% RSLogix 500 project Sample1.RSS, saved by version 9.00.00.04 %
PROJECT "SAMPLE1"    % processor: Bul.1763 MicroLogix 1100 Series A %

PROGRAM FILES
  LAD 2 "MAIN"  21 rungs
  LAD 3 "D INPUT"  11 rungs
  LAD 4 "A INPUT"  66 rungs
  LAD 5 "D OUTPUT"  8 rungs
  LAD 6 "A OUTPUT"  21 rungs
  LAD 7 "ALARMS"  598 rungs
  LAD 8 "HMI IO"  323 rungs
  LAD 9 "LOOPS"  21 rungs
  LAD 10 "CONTROL"  80 rungs

DATA FILES
  O0 OUTPUT  4 elements
  I1 INPUT  6 elements
  S2 STATUS  66 elements
  B3 BINARY  100 elements
  T4 TIMER  256 elements
  C5 COUNTER  1 elements
  R6 CONTROL  1 elements
  N7 INTEGER  256 elements
  F8 FLOAT  249 elements
  B9 ALARMS  40 elements
  F10 F-SETPTS 1  256 elements
  N11 N-SETPTS 1  256 elements
  N12 PIDBLOCKS1  233 elements
  N13 DONOTTOUCH  128 elements
  N14 PIDBLOCKS2  233 elements
  N15 PIDBLOCKS3  143 elements
  B16 SYSCTRLS  10 elements
  T17 TIMERS 2  10 elements
  F18 F-SETPTS 2  93 elements
  N19 N-SETPTS 2  6 elements
  N20 MB_CFG  1 elements
  N21 MB_BIN  46 elements
  F22 MB_FLT1  256 elements
  F23 MB_FLT2  256 elements
  F24 MB_FLT3  256 elements
  F25 MB_FLT4  256 elements
  F26 MB_FLT5  256 elements
  F27 MB_FLT6  256 elements
  F28 MB_FLT7  256 elements
  F29 LAST_VAL1  256 elements
  F30 LAST_VAL2  256 elements
  F31 LAST_VAL3  256 elements
  N90 CH1 Diag  256 elements
  N91 CH0 Diag  32 elements

LADDER 2 "MAIN"
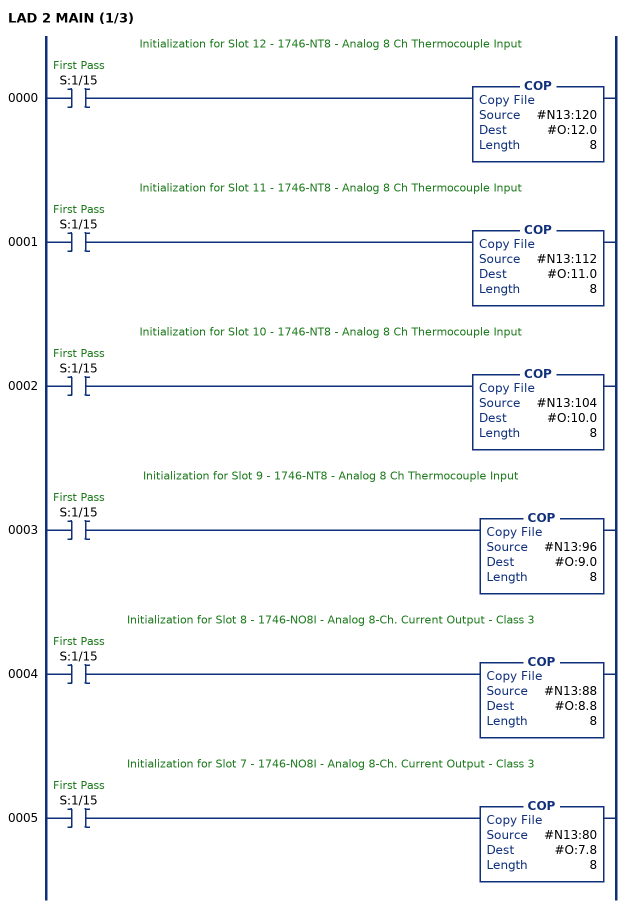
% Rung: 0 %
% Initialization for Slot 12 - 1746-NT8 - Analog 8 Ch Thermocouple Input %
SOR XIC S:1/15 COP #N13:120 #O:12.0 8 EOR
%   S:1/15  "First Pass" %
% Rung: 1 %
% Initialization for Slot 11 - 1746-NT8 - Analog 8 Ch Thermocouple Input %
SOR XIC S:1/15 COP #N13:112 #O:11.0 8 EOR
%   S:1/15  "First Pass" %
% Rung: 2 %
% Initialization for Slot 10 - 1746-NT8 - Analog 8 Ch Thermocouple Input %
SOR XIC S:1/15 COP #N13:104 #O:10.0 8 EOR
%   S:1/15  "First Pass" %
% Rung: 3 %
% Initialization for Slot 9 - 1746-NT8 - Analog 8 Ch Thermocouple Input %
SOR XIC S:1/15 COP #N13:96 #O:9.0 8 EOR
%   S:1/15  "First Pass" %
% Rung: 4 %
% Initialization for Slot 8 - 1746-NO8I - Analog 8-Ch. Current Output - Class 3 %
SOR XIC S:1/15 COP #N13:88 #O:8.8 8 EOR
%   S:1/15  "First Pass" %
% Rung: 5 %
% Initialization for Slot 7 - 1746-NO8I - Analog 8-Ch. Current Output - Class 3 %
SOR XIC S:1/15 COP #N13:80 #O:7.8 8 EOR
%   S:1/15  "First Pass" %

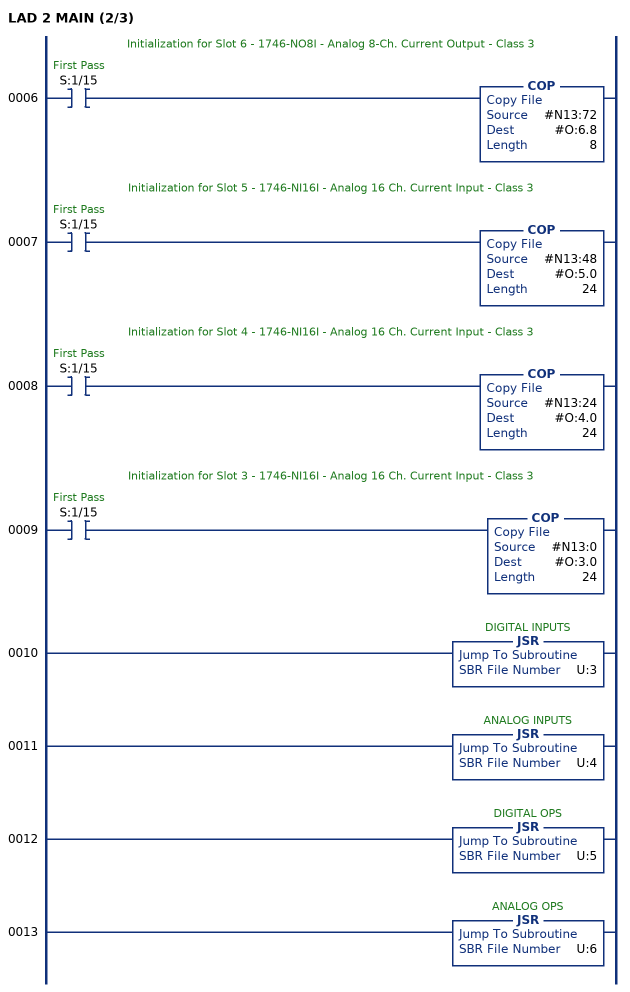
% Rung: 6 %
% Initialization for Slot 6 - 1746-NO8I - Analog 8-Ch. Current Output - Class 3 %
SOR XIC S:1/15 COP #N13:72 #O:6.8 8 EOR
%   S:1/15  "First Pass" %
% Rung: 7 %
% Initialization for Slot 5 - 1746-NI16I - Analog 16 Ch. Current Input - Class 3 %
SOR XIC S:1/15 COP #N13:48 #O:5.0 24 EOR
%   S:1/15  "First Pass" %
% Rung: 8 %
% Initialization for Slot 4 - 1746-NI16I - Analog 16 Ch. Current Input - Class 3 %
SOR XIC S:1/15 COP #N13:24 #O:4.0 24 EOR
%   S:1/15  "First Pass" %
% Rung: 9 %
% Initialization for Slot 3 - 1746-NI16I - Analog 16 Ch. Current Input - Class 3 %
SOR XIC S:1/15 COP #N13:0 #O:3.0 24 EOR
%   S:1/15  "First Pass" %
% Rung: 10 %
SOR JSR U:3 EOR
%   U:3  "DIGITAL INPUTS" %
% Rung: 11 %
SOR JSR U:4 EOR
%   U:4  "ANALOG INPUTS" %
% Rung: 12 %
SOR JSR U:5 EOR
%   U:5  "DIGITAL OPS" %
% Rung: 13 %
SOR JSR U:6 EOR
%   U:6  "ANALOG OPS" %

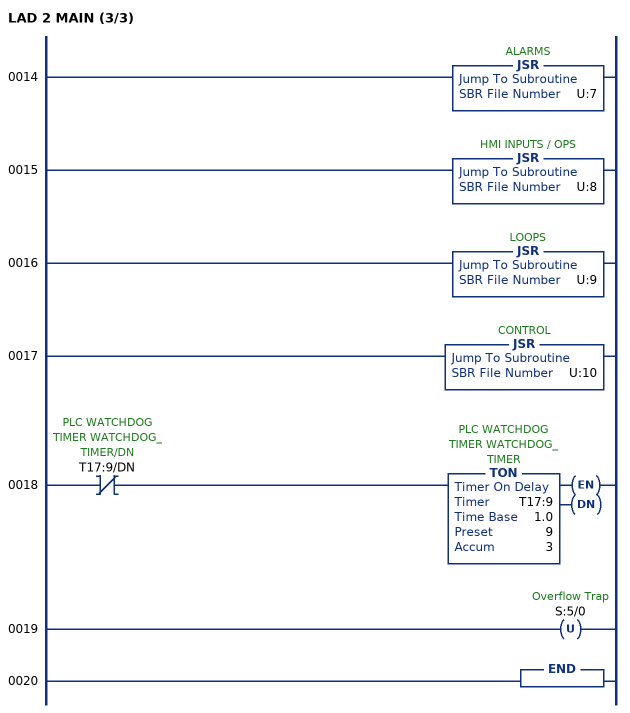
% Rung: 14 %
SOR JSR U:7 EOR
%   U:7  "ALARMS" %
% Rung: 15 %
SOR JSR U:8 EOR
%   U:8  "HMI INPUTS / OPS" %
% Rung: 16 %
SOR JSR U:9 EOR
%   U:9  "LOOPS" %
% Rung: 17 %
SOR JSR U:10 EOR
%   U:10  "CONTROL" %
% Rung: 18 %
SOR XIO T17:9/DN TON T17:9 1.0 9 3 EOR
%   T17:9  WATCHDOG_TIMER  "PLC WATCHDOG TIMER" %
% Rung: 19 %
SOR OTU S:5/0 EOR
%   S:5/0  "Overflow Trap" %
% Rung: 20 %
SOR END EOR

LADDER 3 "D INPUT"
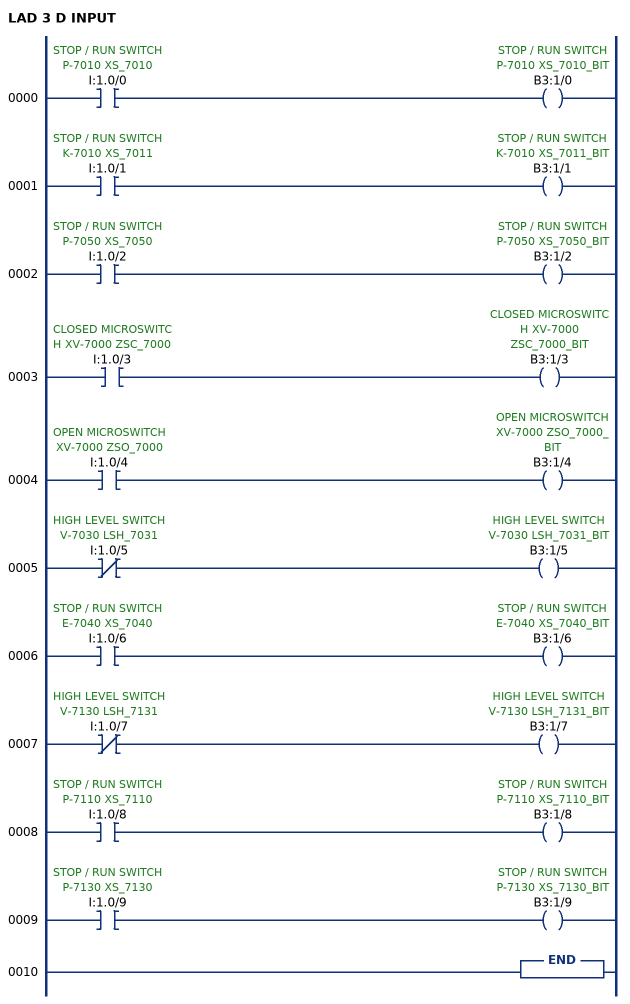
% Rung: 0 %
SOR XIC I:1.0/0 OTE B3:1/0 EOR
%   I:1.0/0  XS_7010  "STOP / RUN SWITCH P-7010" %
%   B3:1/0  XS_7010_BIT  "STOP / RUN SWITCH P-7010" %
% Rung: 1 %
SOR XIC I:1.0/1 OTE B3:1/1 EOR
%   I:1.0/1  XS_7011  "STOP / RUN SWITCH K-7010" %
%   B3:1/1  XS_7011_BIT  "STOP / RUN SWITCH K-7010" %
% Rung: 2 %
SOR XIC I:1.0/2 OTE B3:1/2 EOR
%   I:1.0/2  XS_7050  "STOP / RUN SWITCH P-7050" %
%   B3:1/2  XS_7050_BIT  "STOP / RUN SWITCH P-7050" %
% Rung: 3 %
SOR XIC I:1.0/3 OTE B3:1/3 EOR
%   I:1.0/3  ZSC_7000  "CLOSED MICROSWITCH XV-7000" %
%   B3:1/3  ZSC_7000_BIT  "CLOSED MICROSWITCH XV-7000" %
% Rung: 4 %
SOR XIC I:1.0/4 OTE B3:1/4 EOR
%   I:1.0/4  ZSO_7000  "OPEN MICROSWITCH XV-7000" %
%   B3:1/4  ZSO_7000_BIT  "OPEN MICROSWITCH XV-7000" %
% Rung: 5 %
SOR XIO I:1.0/5 OTE B3:1/5 EOR
%   I:1.0/5  LSH_7031  "HIGH LEVEL SWITCH V-7030" %
%   B3:1/5  LSH_7031_BIT  "HIGH LEVEL SWITCH V-7030" %
% Rung: 6 %
SOR XIC I:1.0/6 OTE B3:1/6 EOR
%   I:1.0/6  XS_7040  "STOP / RUN SWITCH E-7040" %
%   B3:1/6  XS_7040_BIT  "STOP / RUN SWITCH E-7040" %
% Rung: 7 %
SOR XIO I:1.0/7 OTE B3:1/7 EOR
%   I:1.0/7  LSH_7131  "HIGH LEVEL SWITCH V-7130" %
%   B3:1/7  LSH_7131_BIT  "HIGH LEVEL SWITCH V-7130" %
% Rung: 8 %
SOR XIC I:1.0/8 OTE B3:1/8 EOR
%   I:1.0/8  XS_7110  "STOP / RUN SWITCH P-7110" %
%   B3:1/8  XS_7110_BIT  "STOP / RUN SWITCH P-7110" %
% Rung: 9 %
SOR XIC I:1.0/9 OTE B3:1/9 EOR
%   I:1.0/9  XS_7130  "STOP / RUN SWITCH P-7130" %
%   B3:1/9  XS_7130_BIT  "STOP / RUN SWITCH P-7130" %
% Rung: 10 %
SOR END EOR

LADDER 4 "A INPUT"
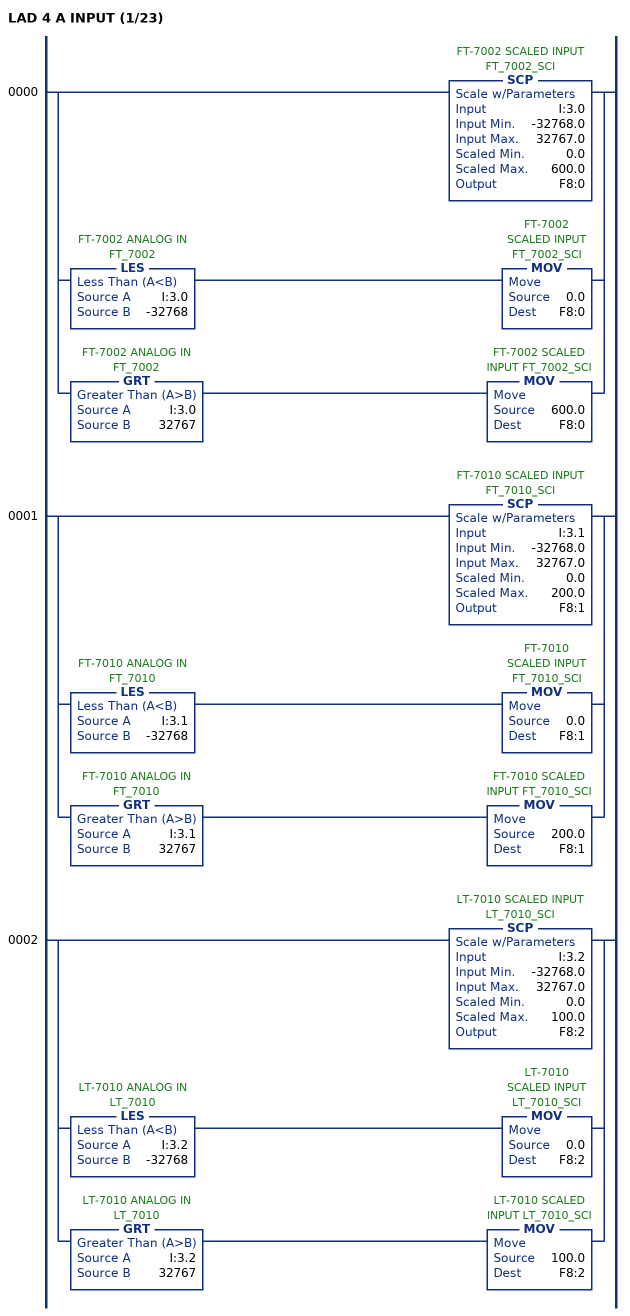
% Rung: 0 %
SOR BST SCP I:3.0 -32768.0 32767.0 0.0 600.0 F8:0 NXB LES I:3.0 -32768 MOV 0.0 F8:0 NXB GRT I:3.0 32767 MOV 600.0 F8:0 BND EOR
%   I:3.0  FT_7002  "FT-7002 ANALOG IN" %
%   F8:0  FT_7002_SCI  "FT-7002 SCALED INPUT" %
% Rung: 1 %
SOR BST SCP I:3.1 -32768.0 32767.0 0.0 200.0 F8:1 NXB LES I:3.1 -32768 MOV 0.0 F8:1 NXB GRT I:3.1 32767 MOV 200.0 F8:1 BND EOR
%   I:3.1  FT_7010  "FT-7010 ANALOG IN" %
%   F8:1  FT_7010_SCI  "FT-7010 SCALED INPUT" %
% Rung: 2 %
SOR BST SCP I:3.2 -32768.0 32767.0 0.0 100.0 F8:2 NXB LES I:3.2 -32768 MOV 0.0 F8:2 NXB GRT I:3.2 32767 MOV 100.0 F8:2 BND EOR
%   I:3.2  LT_7010  "LT-7010 ANALOG IN" %
%   F8:2  LT_7010_SCI  "LT-7010 SCALED INPUT" %

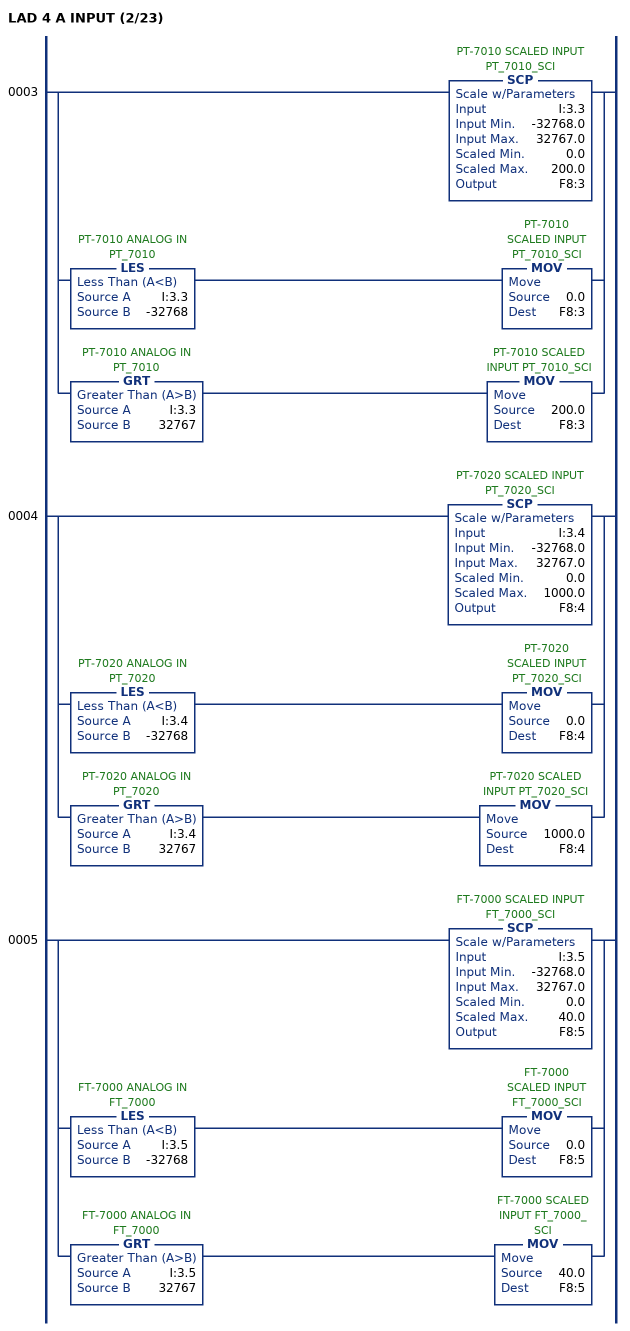
% Rung: 3 %
SOR BST SCP I:3.3 -32768.0 32767.0 0.0 200.0 F8:3 NXB LES I:3.3 -32768 MOV 0.0 F8:3 NXB GRT I:3.3 32767 MOV 200.0 F8:3 BND EOR
%   I:3.3  PT_7010  "PT-7010 ANALOG IN" %
%   F8:3  PT_7010_SCI  "PT-7010 SCALED INPUT" %
% Rung: 4 %
SOR BST SCP I:3.4 -32768.0 32767.0 0.0 1000.0 F8:4 NXB LES I:3.4 -32768 MOV 0.0 F8:4 NXB GRT I:3.4 32767 MOV 1000.0 F8:4 BND EOR
%   I:3.4  PT_7020  "PT-7020 ANALOG IN" %
%   F8:4  PT_7020_SCI  "PT-7020 SCALED INPUT" %
% Rung: 5 %
SOR BST SCP I:3.5 -32768.0 32767.0 0.0 40.0 F8:5 NXB LES I:3.5 -32768 MOV 0.0 F8:5 NXB GRT I:3.5 32767 MOV 40.0 F8:5 BND EOR
%   I:3.5  FT_7000  "FT-7000 ANALOG IN" %
%   F8:5  FT_7000_SCI  "FT-7000 SCALED INPUT" %

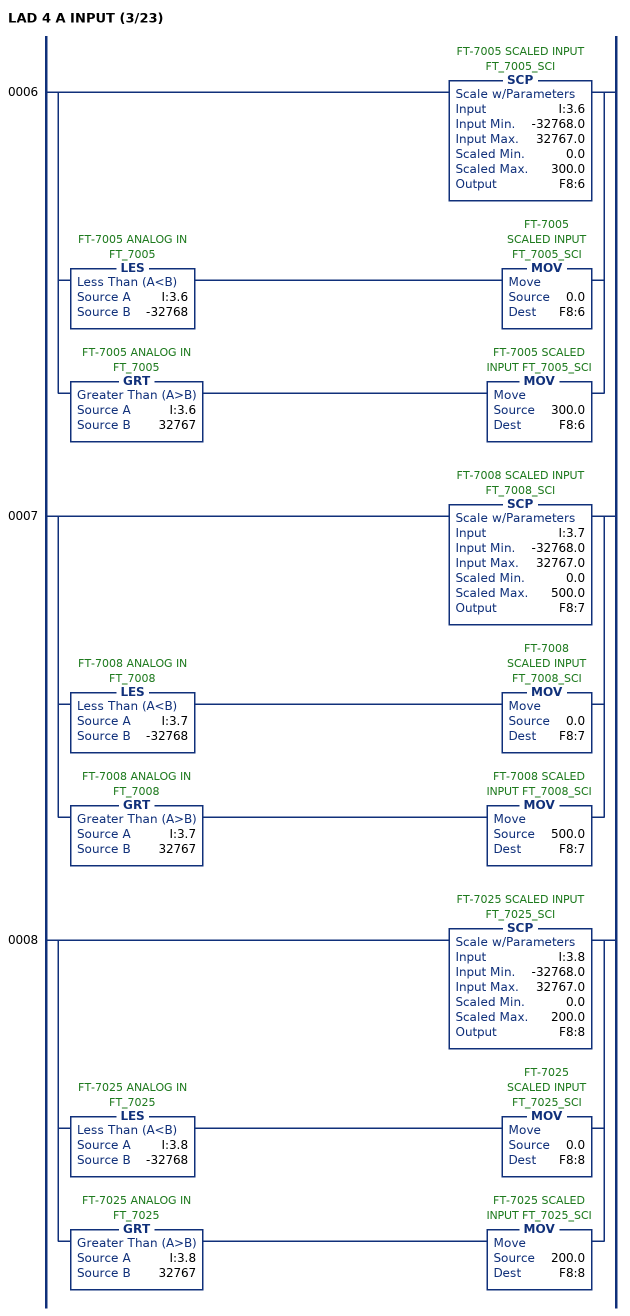
% Rung: 6 %
SOR BST SCP I:3.6 -32768.0 32767.0 0.0 300.0 F8:6 NXB LES I:3.6 -32768 MOV 0.0 F8:6 NXB GRT I:3.6 32767 MOV 300.0 F8:6 BND EOR
%   I:3.6  FT_7005  "FT-7005 ANALOG IN" %
%   F8:6  FT_7005_SCI  "FT-7005 SCALED INPUT" %
% Rung: 7 %
SOR BST SCP I:3.7 -32768.0 32767.0 0.0 500.0 F8:7 NXB LES I:3.7 -32768 MOV 0.0 F8:7 NXB GRT I:3.7 32767 MOV 500.0 F8:7 BND EOR
%   I:3.7  FT_7008  "FT-7008 ANALOG IN" %
%   F8:7  FT_7008_SCI  "FT-7008 SCALED INPUT" %
% Rung: 8 %
SOR BST SCP I:3.8 -32768.0 32767.0 0.0 200.0 F8:8 NXB LES I:3.8 -32768 MOV 0.0 F8:8 NXB GRT I:3.8 32767 MOV 200.0 F8:8 BND EOR
%   I:3.8  FT_7025  "FT-7025 ANALOG IN" %
%   F8:8  FT_7025_SCI  "FT-7025 SCALED INPUT" %

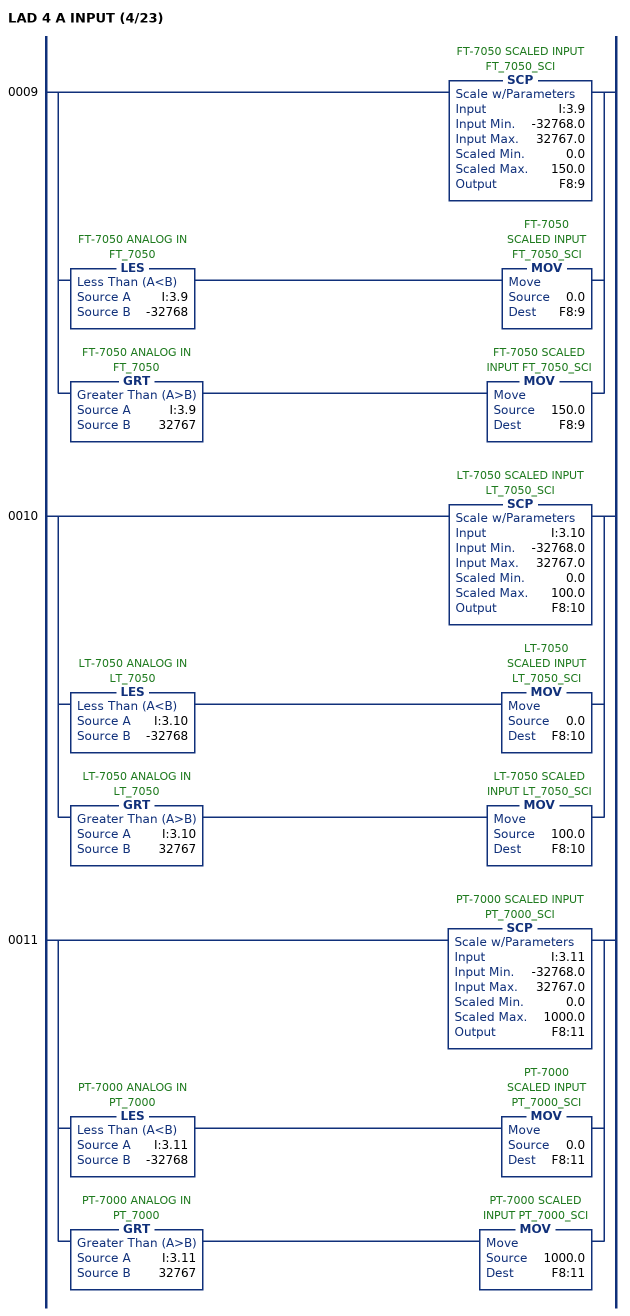
% Rung: 9 %
SOR BST SCP I:3.9 -32768.0 32767.0 0.0 150.0 F8:9 NXB LES I:3.9 -32768 MOV 0.0 F8:9 NXB GRT I:3.9 32767 MOV 150.0 F8:9 BND EOR
%   I:3.9  FT_7050  "FT-7050 ANALOG IN" %
%   F8:9  FT_7050_SCI  "FT-7050 SCALED INPUT" %
% Rung: 10 %
SOR BST SCP I:3.10 -32768.0 32767.0 0.0 100.0 F8:10 NXB LES I:3.10 -32768 MOV 0.0 F8:10 NXB GRT I:3.10 32767 MOV 100.0 F8:10 BND EOR
%   I:3.10  LT_7050  "LT-7050 ANALOG IN" %
%   F8:10  LT_7050_SCI  "LT-7050 SCALED INPUT" %
% Rung: 11 %
SOR BST SCP I:3.11 -32768.0 32767.0 0.0 1000.0 F8:11 NXB LES I:3.11 -32768 MOV 0.0 F8:11 NXB GRT I:3.11 32767 MOV 1000.0 F8:11 BND EOR
%   I:3.11  PT_7000  "PT-7000 ANALOG IN" %
%   F8:11  PT_7000_SCI  "PT-7000 SCALED INPUT" %

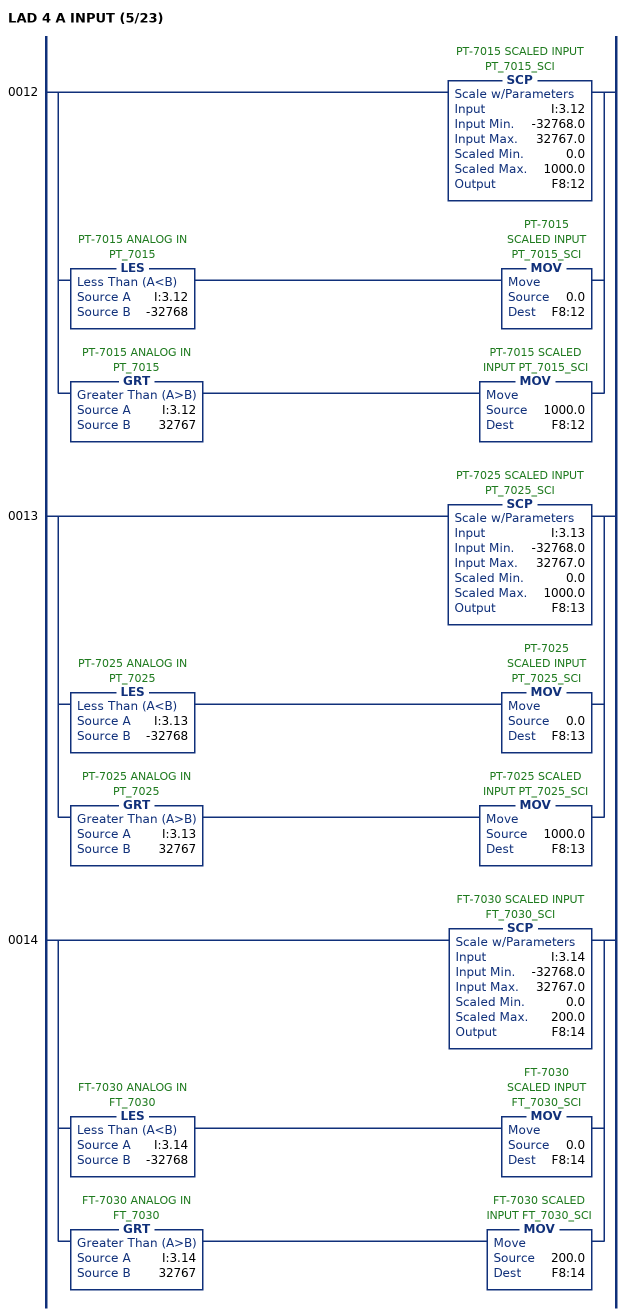
% Rung: 12 %
SOR BST SCP I:3.12 -32768.0 32767.0 0.0 1000.0 F8:12 NXB LES I:3.12 -32768 MOV 0.0 F8:12 NXB GRT I:3.12 32767 MOV 1000.0 F8:12 BND EOR
%   I:3.12  PT_7015  "PT-7015 ANALOG IN" %
%   F8:12  PT_7015_SCI  "PT-7015 SCALED INPUT" %
% Rung: 13 %
SOR BST SCP I:3.13 -32768.0 32767.0 0.0 1000.0 F8:13 NXB LES I:3.13 -32768 MOV 0.0 F8:13 NXB GRT I:3.13 32767 MOV 1000.0 F8:13 BND EOR
%   I:3.13  PT_7025  "PT-7025 ANALOG IN" %
%   F8:13  PT_7025_SCI  "PT-7025 SCALED INPUT" %
% Rung: 14 %
SOR BST SCP I:3.14 -32768.0 32767.0 0.0 200.0 F8:14 NXB LES I:3.14 -32768 MOV 0.0 F8:14 NXB GRT I:3.14 32767 MOV 200.0 F8:14 BND EOR
%   I:3.14  FT_7030  "FT-7030 ANALOG IN" %
%   F8:14  FT_7030_SCI  "FT-7030 SCALED INPUT" %

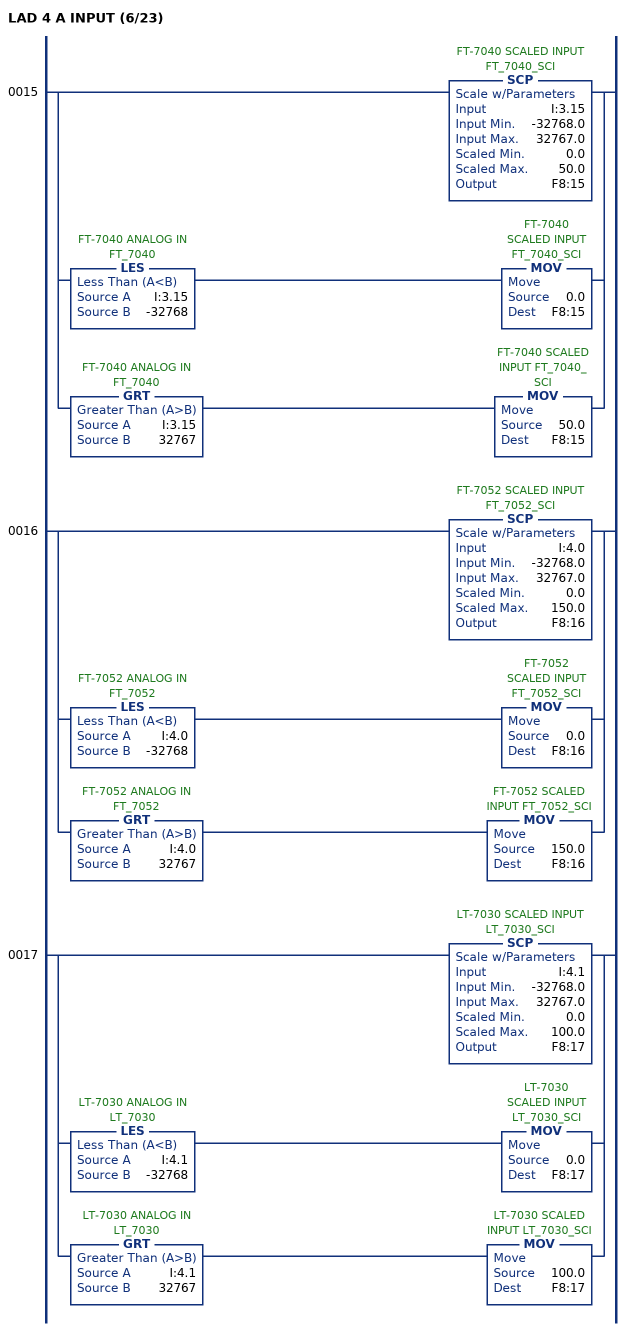
% Rung: 15 %
SOR BST SCP I:3.15 -32768.0 32767.0 0.0 50.0 F8:15 NXB LES I:3.15 -32768 MOV 0.0 F8:15 NXB GRT I:3.15 32767 MOV 50.0 F8:15 BND EOR
%   I:3.15  FT_7040  "FT-7040 ANALOG IN" %
%   F8:15  FT_7040_SCI  "FT-7040 SCALED INPUT" %
% Rung: 16 %
SOR BST SCP I:4.0 -32768.0 32767.0 0.0 150.0 F8:16 NXB LES I:4.0 -32768 MOV 0.0 F8:16 NXB GRT I:4.0 32767 MOV 150.0 F8:16 BND EOR
%   I:4.0  FT_7052  "FT-7052 ANALOG IN" %
%   F8:16  FT_7052_SCI  "FT-7052 SCALED INPUT" %
% Rung: 17 %
SOR BST SCP I:4.1 -32768.0 32767.0 0.0 100.0 F8:17 NXB LES I:4.1 -32768 MOV 0.0 F8:17 NXB GRT I:4.1 32767 MOV 100.0 F8:17 BND EOR
%   I:4.1  LT_7030  "LT-7030 ANALOG IN" %
%   F8:17  LT_7030_SCI  "LT-7030 SCALED INPUT" %

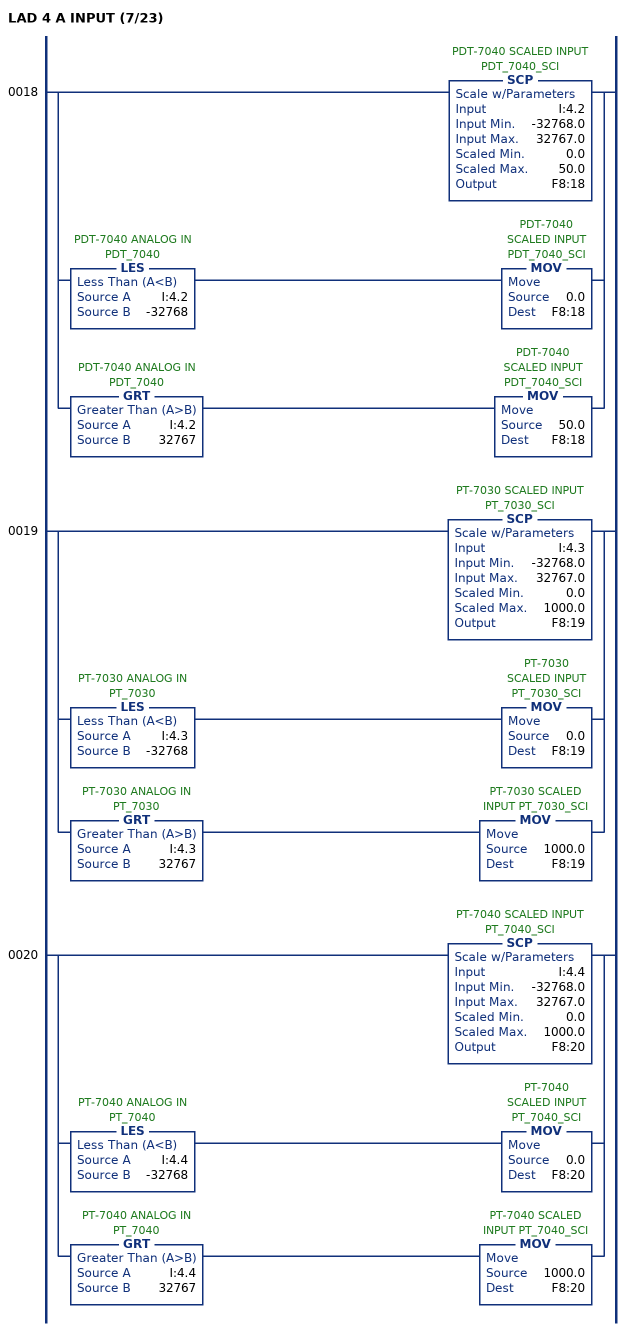
% Rung: 18 %
SOR BST SCP I:4.2 -32768.0 32767.0 0.0 50.0 F8:18 NXB LES I:4.2 -32768 MOV 0.0 F8:18 NXB GRT I:4.2 32767 MOV 50.0 F8:18 BND EOR
%   I:4.2  PDT_7040  "PDT-7040 ANALOG IN" %
%   F8:18  PDT_7040_SCI  "PDT-7040 SCALED INPUT" %
% Rung: 19 %
SOR BST SCP I:4.3 -32768.0 32767.0 0.0 1000.0 F8:19 NXB LES I:4.3 -32768 MOV 0.0 F8:19 NXB GRT I:4.3 32767 MOV 1000.0 F8:19 BND EOR
%   I:4.3  PT_7030  "PT-7030 ANALOG IN" %
%   F8:19  PT_7030_SCI  "PT-7030 SCALED INPUT" %
% Rung: 20 %
SOR BST SCP I:4.4 -32768.0 32767.0 0.0 1000.0 F8:20 NXB LES I:4.4 -32768 MOV 0.0 F8:20 NXB GRT I:4.4 32767 MOV 1000.0 F8:20 BND EOR
%   I:4.4  PT_7040  "PT-7040 ANALOG IN" %
%   F8:20  PT_7040_SCI  "PT-7040 SCALED INPUT" %

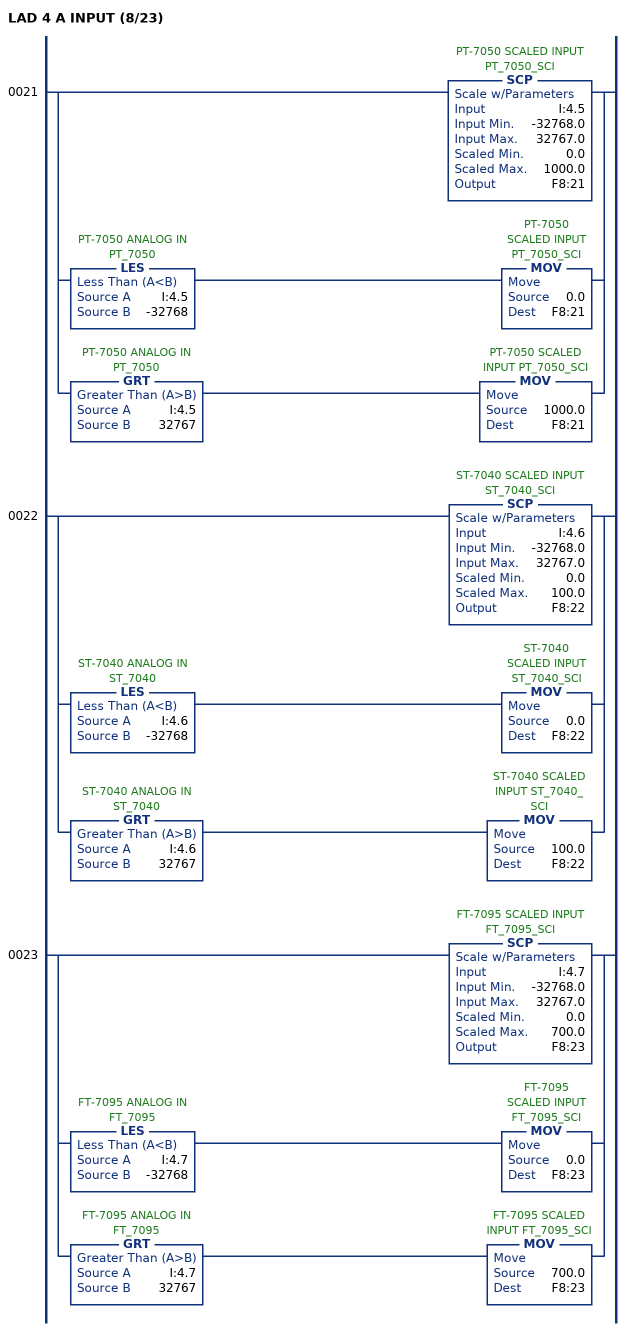
% Rung: 21 %
SOR BST SCP I:4.5 -32768.0 32767.0 0.0 1000.0 F8:21 NXB LES I:4.5 -32768 MOV 0.0 F8:21 NXB GRT I:4.5 32767 MOV 1000.0 F8:21 BND EOR
%   I:4.5  PT_7050  "PT-7050 ANALOG IN" %
%   F8:21  PT_7050_SCI  "PT-7050 SCALED INPUT" %
% Rung: 22 %
SOR BST SCP I:4.6 -32768.0 32767.0 0.0 100.0 F8:22 NXB LES I:4.6 -32768 MOV 0.0 F8:22 NXB GRT I:4.6 32767 MOV 100.0 F8:22 BND EOR
%   I:4.6  ST_7040  "ST-7040 ANALOG IN" %
%   F8:22  ST_7040_SCI  "ST-7040 SCALED INPUT" %
% Rung: 23 %
SOR BST SCP I:4.7 -32768.0 32767.0 0.0 700.0 F8:23 NXB LES I:4.7 -32768 MOV 0.0 F8:23 NXB GRT I:4.7 32767 MOV 700.0 F8:23 BND EOR
%   I:4.7  FT_7095  "FT-7095 ANALOG IN" %
%   F8:23  FT_7095_SCI  "FT-7095 SCALED INPUT" %

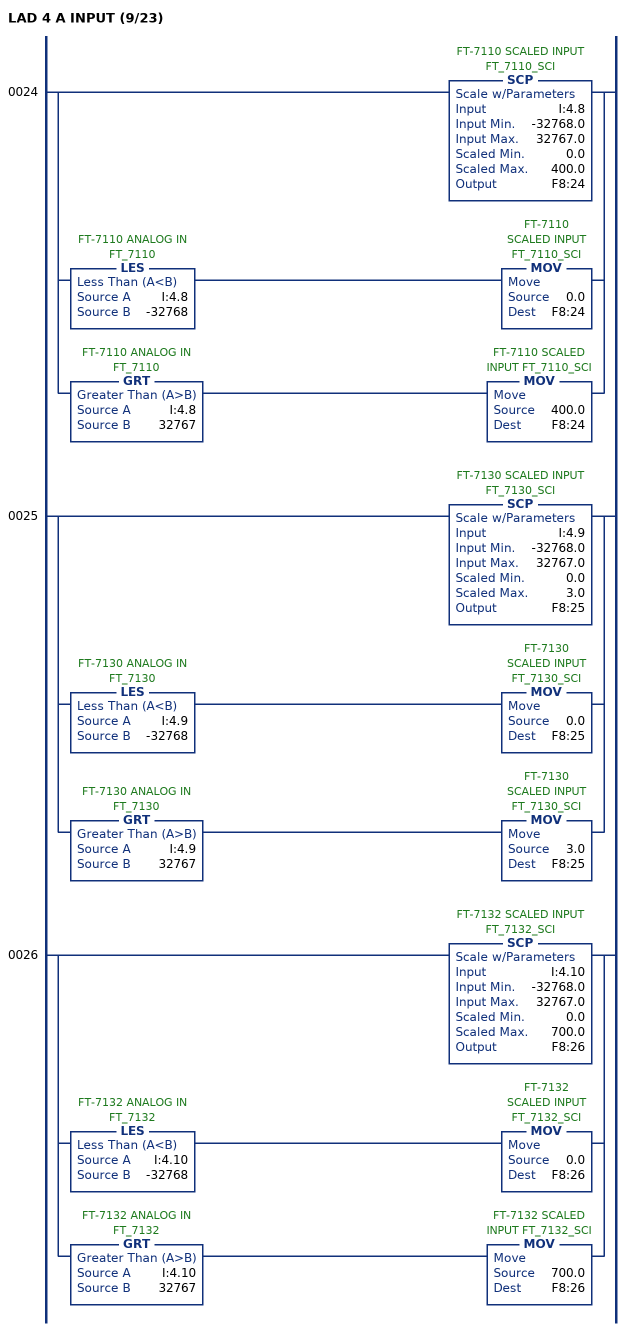
% Rung: 24 %
SOR BST SCP I:4.8 -32768.0 32767.0 0.0 400.0 F8:24 NXB LES I:4.8 -32768 MOV 0.0 F8:24 NXB GRT I:4.8 32767 MOV 400.0 F8:24 BND EOR
%   I:4.8  FT_7110  "FT-7110 ANALOG IN" %
%   F8:24  FT_7110_SCI  "FT-7110 SCALED INPUT" %
% Rung: 25 %
SOR BST SCP I:4.9 -32768.0 32767.0 0.0 3.0 F8:25 NXB LES I:4.9 -32768 MOV 0.0 F8:25 NXB GRT I:4.9 32767 MOV 3.0 F8:25 BND EOR
%   I:4.9  FT_7130  "FT-7130 ANALOG IN" %
%   F8:25  FT_7130_SCI  "FT-7130 SCALED INPUT" %
% Rung: 26 %
SOR BST SCP I:4.10 -32768.0 32767.0 0.0 700.0 F8:26 NXB LES I:4.10 -32768 MOV 0.0 F8:26 NXB GRT I:4.10 32767 MOV 700.0 F8:26 BND EOR
%   I:4.10  FT_7132  "FT-7132 ANALOG IN" %
%   F8:26  FT_7132_SCI  "FT-7132 SCALED INPUT" %

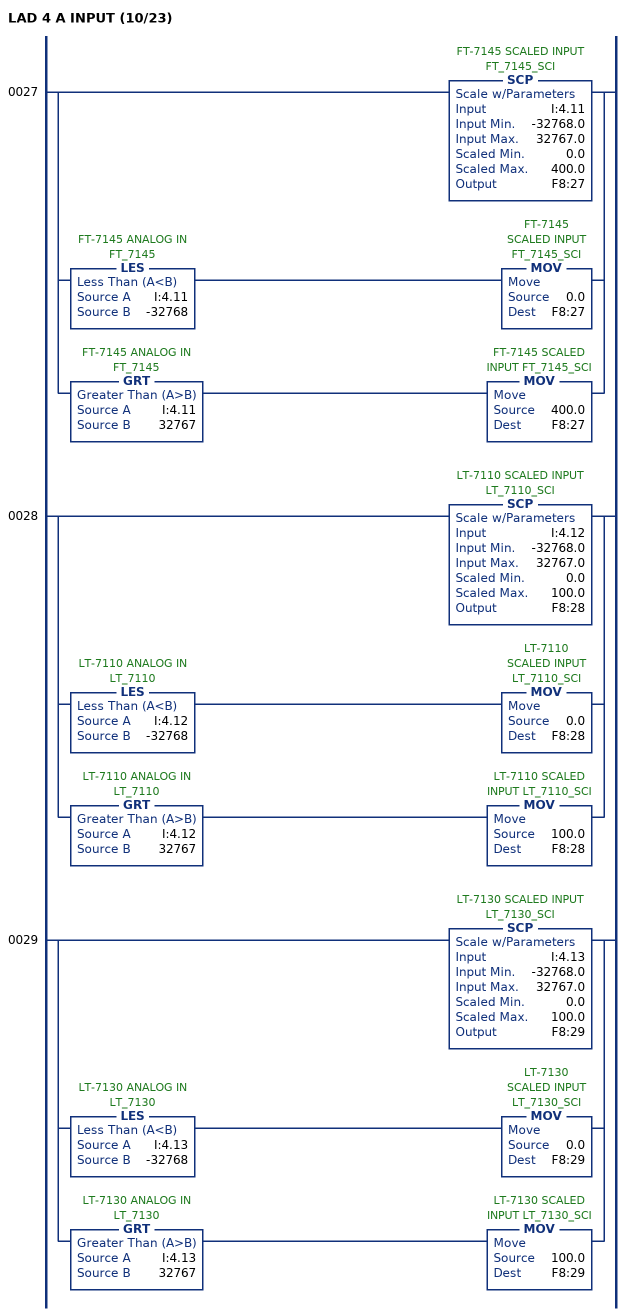
% Rung: 27 %
SOR BST SCP I:4.11 -32768.0 32767.0 0.0 400.0 F8:27 NXB LES I:4.11 -32768 MOV 0.0 F8:27 NXB GRT I:4.11 32767 MOV 400.0 F8:27 BND EOR
%   I:4.11  FT_7145  "FT-7145 ANALOG IN" %
%   F8:27  FT_7145_SCI  "FT-7145 SCALED INPUT" %
% Rung: 28 %
SOR BST SCP I:4.12 -32768.0 32767.0 0.0 100.0 F8:28 NXB LES I:4.12 -32768 MOV 0.0 F8:28 NXB GRT I:4.12 32767 MOV 100.0 F8:28 BND EOR
%   I:4.12  LT_7110  "LT-7110 ANALOG IN" %
%   F8:28  LT_7110_SCI  "LT-7110 SCALED INPUT" %
% Rung: 29 %
SOR BST SCP I:4.13 -32768.0 32767.0 0.0 100.0 F8:29 NXB LES I:4.13 -32768 MOV 0.0 F8:29 NXB GRT I:4.13 32767 MOV 100.0 F8:29 BND EOR
%   I:4.13  LT_7130  "LT-7130 ANALOG IN" %
%   F8:29  LT_7130_SCI  "LT-7130 SCALED INPUT" %

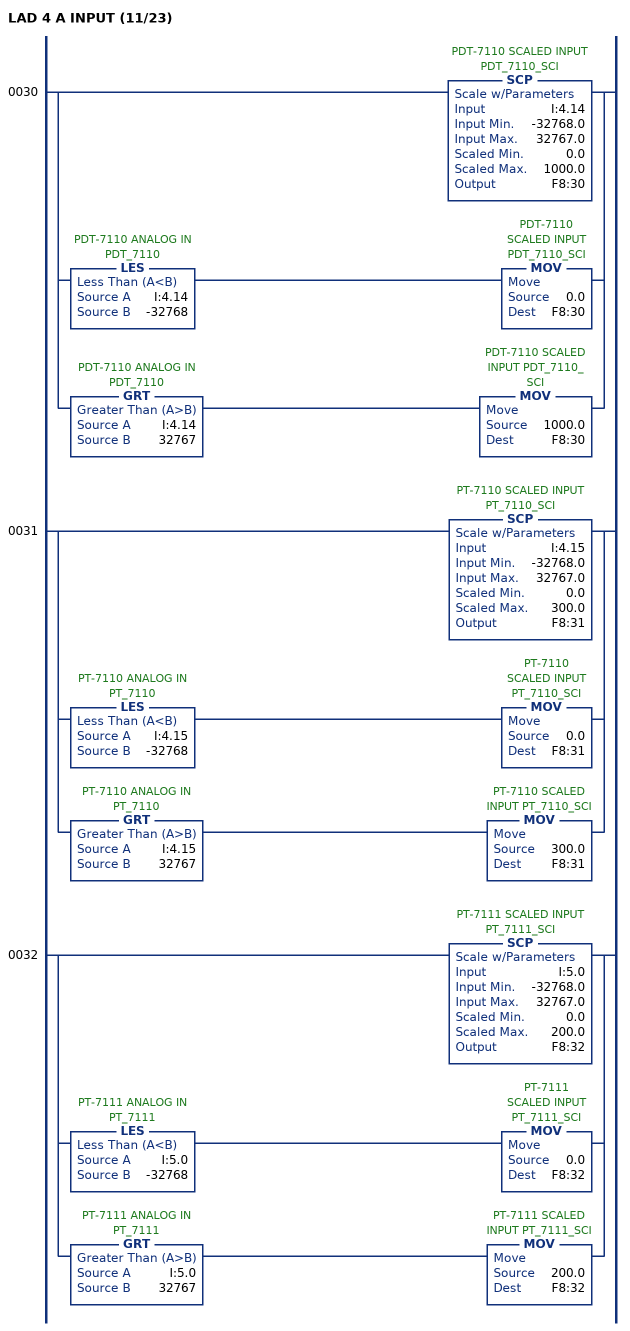
% Rung: 30 %
SOR BST SCP I:4.14 -32768.0 32767.0 0.0 1000.0 F8:30 NXB LES I:4.14 -32768 MOV 0.0 F8:30 NXB GRT I:4.14 32767 MOV 1000.0 F8:30 BND EOR
%   I:4.14  PDT_7110  "PDT-7110 ANALOG IN" %
%   F8:30  PDT_7110_SCI  "PDT-7110 SCALED INPUT" %
% Rung: 31 %
SOR BST SCP I:4.15 -32768.0 32767.0 0.0 300.0 F8:31 NXB LES I:4.15 -32768 MOV 0.0 F8:31 NXB GRT I:4.15 32767 MOV 300.0 F8:31 BND EOR
%   I:4.15  PT_7110  "PT-7110 ANALOG IN" %
%   F8:31  PT_7110_SCI  "PT-7110 SCALED INPUT" %
% Rung: 32 %
SOR BST SCP I:5.0 -32768.0 32767.0 0.0 200.0 F8:32 NXB LES I:5.0 -32768 MOV 0.0 F8:32 NXB GRT I:5.0 32767 MOV 200.0 F8:32 BND EOR
%   I:5.0  PT_7111  "PT-7111 ANALOG IN" %
%   F8:32  PT_7111_SCI  "PT-7111 SCALED INPUT" %

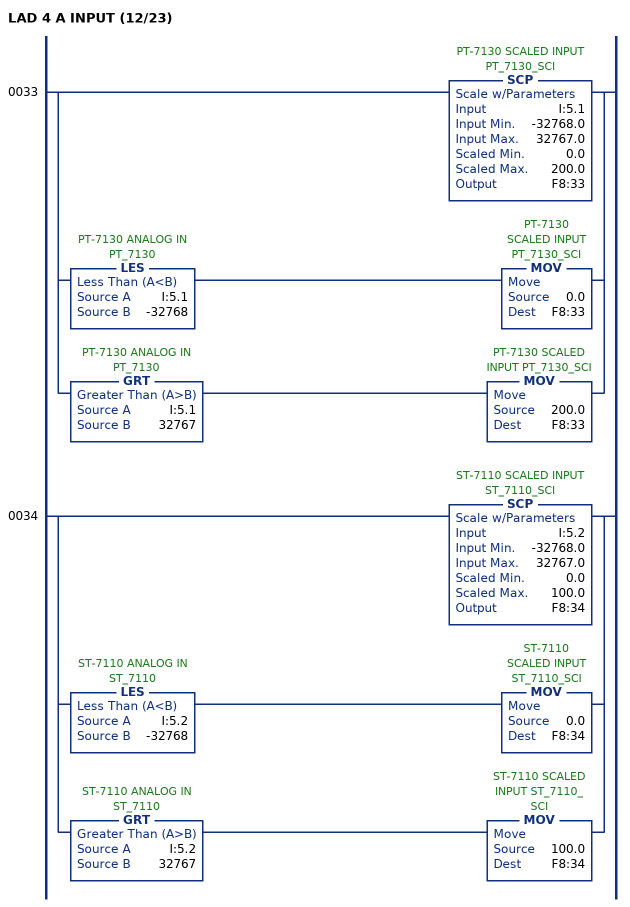
% Rung: 33 %
SOR BST SCP I:5.1 -32768.0 32767.0 0.0 200.0 F8:33 NXB LES I:5.1 -32768 MOV 0.0 F8:33 NXB GRT I:5.1 32767 MOV 200.0 F8:33 BND EOR
%   I:5.1  PT_7130  "PT-7130 ANALOG IN" %
%   F8:33  PT_7130_SCI  "PT-7130 SCALED INPUT" %
% Rung: 34 %
SOR BST SCP I:5.2 -32768.0 32767.0 0.0 100.0 F8:34 NXB LES I:5.2 -32768 MOV 0.0 F8:34 NXB GRT I:5.2 32767 MOV 100.0 F8:34 BND EOR
%   I:5.2  ST_7110  "ST-7110 ANALOG IN" %
%   F8:34  ST_7110_SCI  "ST-7110 SCALED INPUT" %

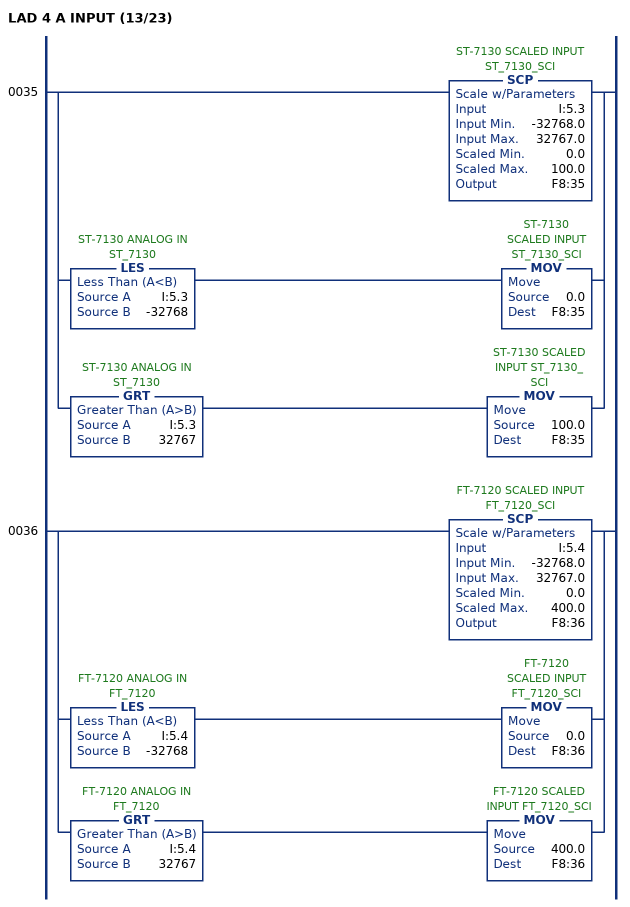
% Rung: 35 %
SOR BST SCP I:5.3 -32768.0 32767.0 0.0 100.0 F8:35 NXB LES I:5.3 -32768 MOV 0.0 F8:35 NXB GRT I:5.3 32767 MOV 100.0 F8:35 BND EOR
%   I:5.3  ST_7130  "ST-7130 ANALOG IN" %
%   F8:35  ST_7130_SCI  "ST-7130 SCALED INPUT" %
% Rung: 36 %
SOR BST SCP I:5.4 -32768.0 32767.0 0.0 400.0 F8:36 NXB LES I:5.4 -32768 MOV 0.0 F8:36 NXB GRT I:5.4 32767 MOV 400.0 F8:36 BND EOR
%   I:5.4  FT_7120  "FT-7120 ANALOG IN" %
%   F8:36  FT_7120_SCI  "FT-7120 SCALED INPUT" %

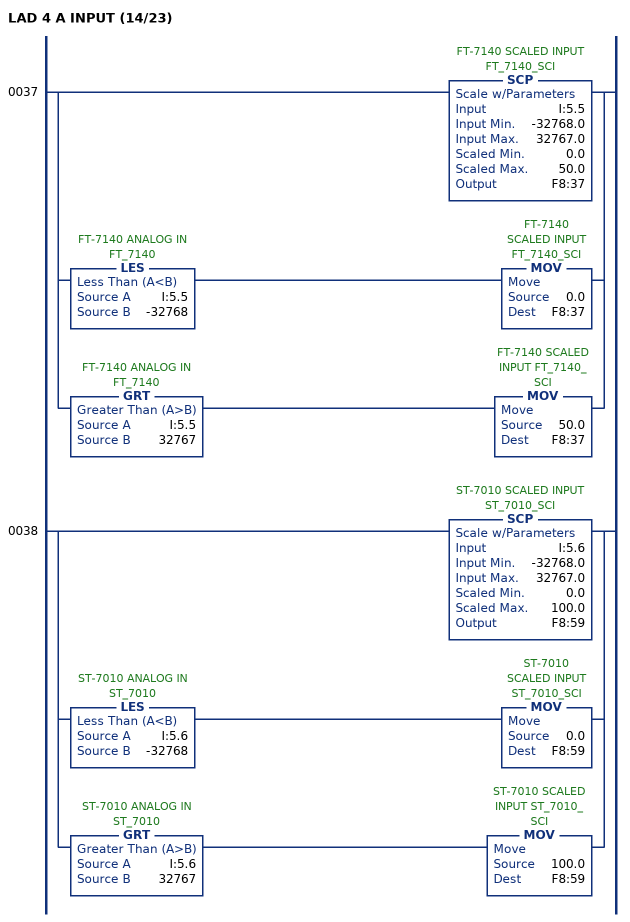
% Rung: 37 %
SOR BST SCP I:5.5 -32768.0 32767.0 0.0 50.0 F8:37 NXB LES I:5.5 -32768 MOV 0.0 F8:37 NXB GRT I:5.5 32767 MOV 50.0 F8:37 BND EOR
%   I:5.5  FT_7140  "FT-7140 ANALOG IN" %
%   F8:37  FT_7140_SCI  "FT-7140 SCALED INPUT" %
% Rung: 38 %
SOR BST SCP I:5.6 -32768.0 32767.0 0.0 100.0 F8:59 NXB LES I:5.6 -32768 MOV 0.0 F8:59 NXB GRT I:5.6 32767 MOV 100.0 F8:59 BND EOR
%   I:5.6  ST_7010  "ST-7010 ANALOG IN" %
%   F8:59  ST_7010_SCI  "ST-7010 SCALED INPUT" %

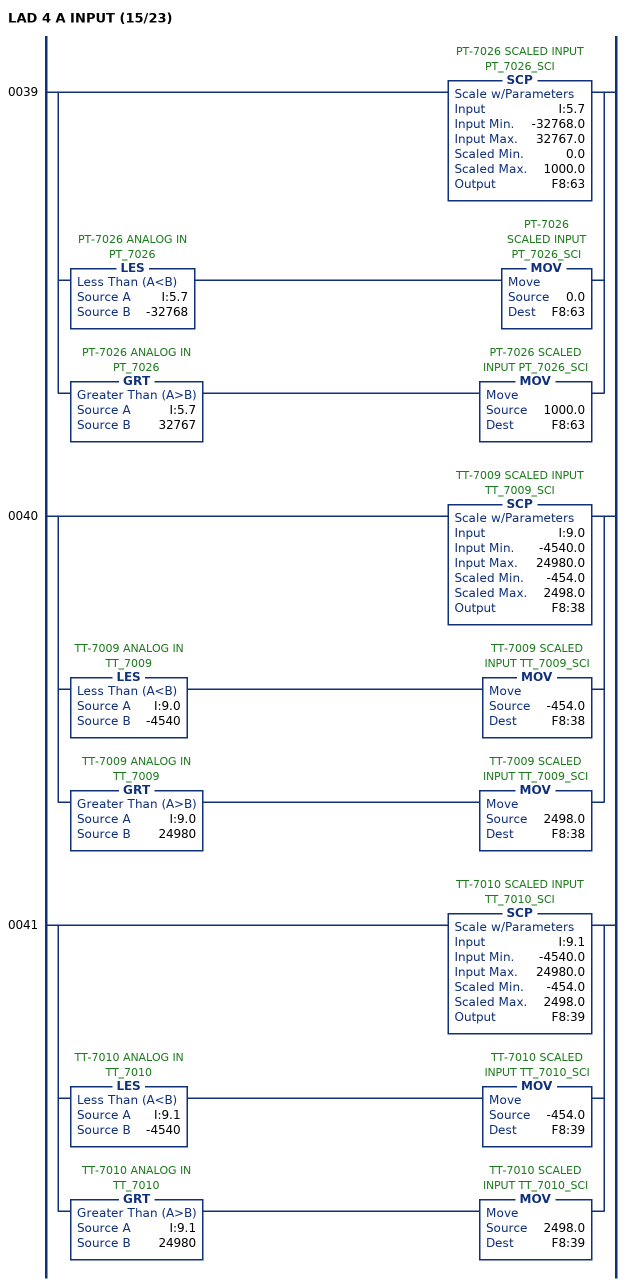
% Rung: 39 %
SOR BST SCP I:5.7 -32768.0 32767.0 0.0 1000.0 F8:63 NXB LES I:5.7 -32768 MOV 0.0 F8:63 NXB GRT I:5.7 32767 MOV 1000.0 F8:63 BND EOR
%   I:5.7  PT_7026  "PT-7026 ANALOG IN" %
%   F8:63  PT_7026_SCI  "PT-7026 SCALED INPUT" %
% Rung: 40 %
SOR BST SCP I:9.0 -4540.0 24980.0 -454.0 2498.0 F8:38 NXB LES I:9.0 -4540 MOV -454.0 F8:38 NXB GRT I:9.0 24980 MOV 2498.0 F8:38 BND EOR
%   I:9.0  TT_7009  "TT-7009 ANALOG IN" %
%   F8:38  TT_7009_SCI  "TT-7009 SCALED INPUT" %
% Rung: 41 %
SOR BST SCP I:9.1 -4540.0 24980.0 -454.0 2498.0 F8:39 NXB LES I:9.1 -4540 MOV -454.0 F8:39 NXB GRT I:9.1 24980 MOV 2498.0 F8:39 BND EOR
%   I:9.1  TT_7010  "TT-7010 ANALOG IN" %
%   F8:39  TT_7010_SCI  "TT-7010 SCALED INPUT" %

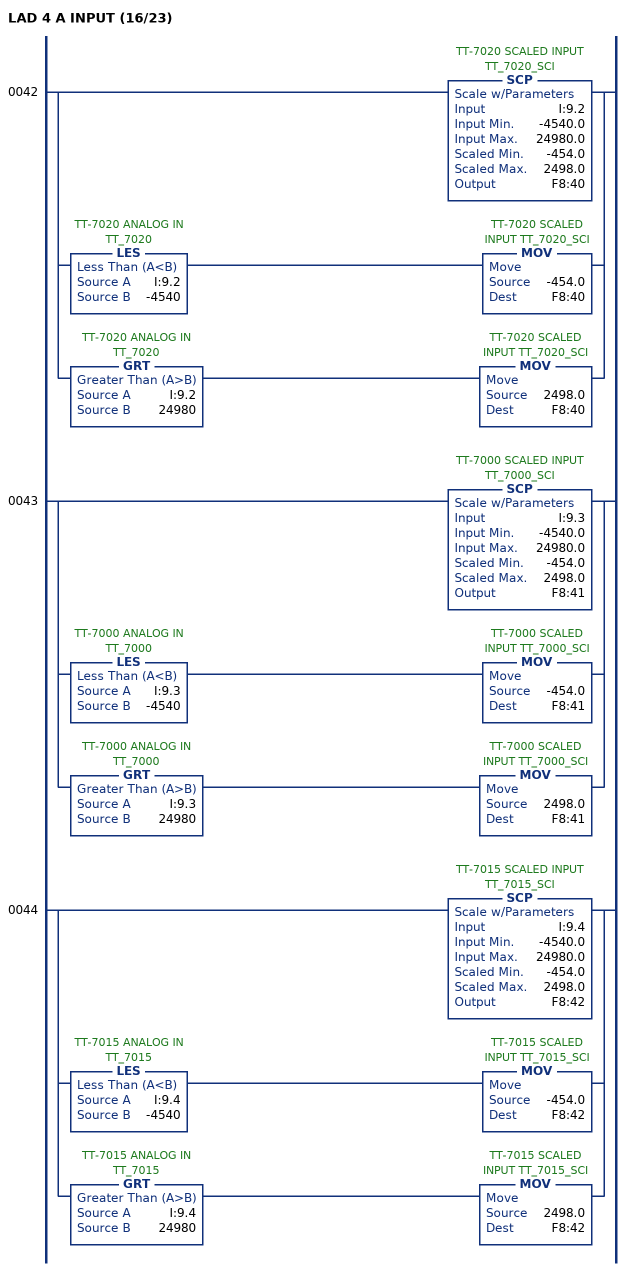
% Rung: 42 %
SOR BST SCP I:9.2 -4540.0 24980.0 -454.0 2498.0 F8:40 NXB LES I:9.2 -4540 MOV -454.0 F8:40 NXB GRT I:9.2 24980 MOV 2498.0 F8:40 BND EOR
%   I:9.2  TT_7020  "TT-7020 ANALOG IN" %
%   F8:40  TT_7020_SCI  "TT-7020 SCALED INPUT" %
% Rung: 43 %
SOR BST SCP I:9.3 -4540.0 24980.0 -454.0 2498.0 F8:41 NXB LES I:9.3 -4540 MOV -454.0 F8:41 NXB GRT I:9.3 24980 MOV 2498.0 F8:41 BND EOR
%   I:9.3  TT_7000  "TT-7000 ANALOG IN" %
%   F8:41  TT_7000_SCI  "TT-7000 SCALED INPUT" %
% Rung: 44 %
SOR BST SCP I:9.4 -4540.0 24980.0 -454.0 2498.0 F8:42 NXB LES I:9.4 -4540 MOV -454.0 F8:42 NXB GRT I:9.4 24980 MOV 2498.0 F8:42 BND EOR
%   I:9.4  TT_7015  "TT-7015 ANALOG IN" %
%   F8:42  TT_7015_SCI  "TT-7015 SCALED INPUT" %

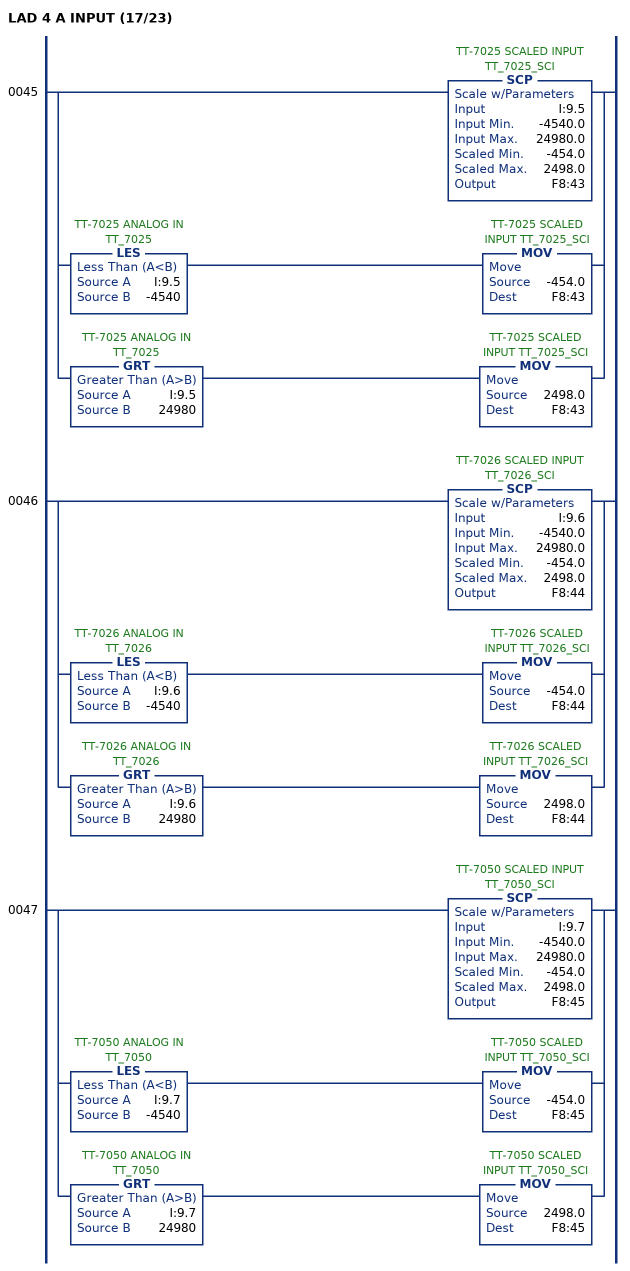
% Rung: 45 %
SOR BST SCP I:9.5 -4540.0 24980.0 -454.0 2498.0 F8:43 NXB LES I:9.5 -4540 MOV -454.0 F8:43 NXB GRT I:9.5 24980 MOV 2498.0 F8:43 BND EOR
%   I:9.5  TT_7025  "TT-7025 ANALOG IN" %
%   F8:43  TT_7025_SCI  "TT-7025 SCALED INPUT" %
% Rung: 46 %
SOR BST SCP I:9.6 -4540.0 24980.0 -454.0 2498.0 F8:44 NXB LES I:9.6 -4540 MOV -454.0 F8:44 NXB GRT I:9.6 24980 MOV 2498.0 F8:44 BND EOR
%   I:9.6  TT_7026  "TT-7026 ANALOG IN" %
%   F8:44  TT_7026_SCI  "TT-7026 SCALED INPUT" %
% Rung: 47 %
SOR BST SCP I:9.7 -4540.0 24980.0 -454.0 2498.0 F8:45 NXB LES I:9.7 -4540 MOV -454.0 F8:45 NXB GRT I:9.7 24980 MOV 2498.0 F8:45 BND EOR
%   I:9.7  TT_7050  "TT-7050 ANALOG IN" %
%   F8:45  TT_7050_SCI  "TT-7050 SCALED INPUT" %

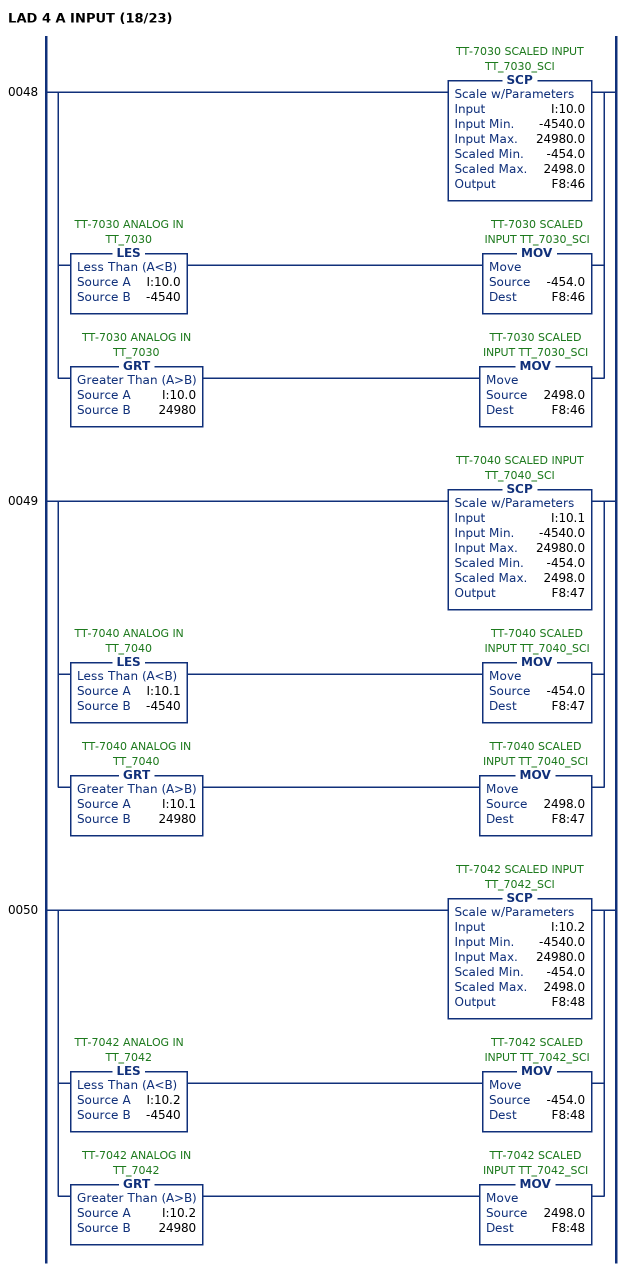
% Rung: 48 %
SOR BST SCP I:10.0 -4540.0 24980.0 -454.0 2498.0 F8:46 NXB LES I:10.0 -4540 MOV -454.0 F8:46 NXB GRT I:10.0 24980 MOV 2498.0 F8:46 BND EOR
%   I:10.0  TT_7030  "TT-7030 ANALOG IN" %
%   F8:46  TT_7030_SCI  "TT-7030 SCALED INPUT" %
% Rung: 49 %
SOR BST SCP I:10.1 -4540.0 24980.0 -454.0 2498.0 F8:47 NXB LES I:10.1 -4540 MOV -454.0 F8:47 NXB GRT I:10.1 24980 MOV 2498.0 F8:47 BND EOR
%   I:10.1  TT_7040  "TT-7040 ANALOG IN" %
%   F8:47  TT_7040_SCI  "TT-7040 SCALED INPUT" %
% Rung: 50 %
SOR BST SCP I:10.2 -4540.0 24980.0 -454.0 2498.0 F8:48 NXB LES I:10.2 -4540 MOV -454.0 F8:48 NXB GRT I:10.2 24980 MOV 2498.0 F8:48 BND EOR
%   I:10.2  TT_7042  "TT-7042 ANALOG IN" %
%   F8:48  TT_7042_SCI  "TT-7042 SCALED INPUT" %

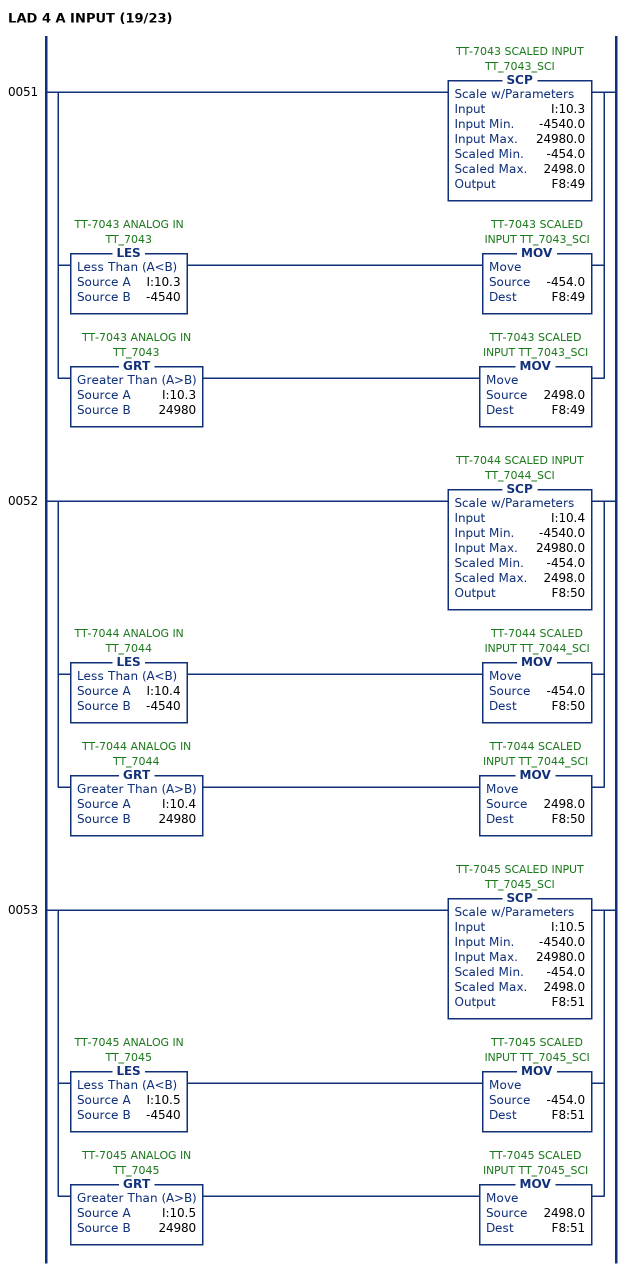
% Rung: 51 %
SOR BST SCP I:10.3 -4540.0 24980.0 -454.0 2498.0 F8:49 NXB LES I:10.3 -4540 MOV -454.0 F8:49 NXB GRT I:10.3 24980 MOV 2498.0 F8:49 BND EOR
%   I:10.3  TT_7043  "TT-7043 ANALOG IN" %
%   F8:49  TT_7043_SCI  "TT-7043 SCALED INPUT" %
% Rung: 52 %
SOR BST SCP I:10.4 -4540.0 24980.0 -454.0 2498.0 F8:50 NXB LES I:10.4 -4540 MOV -454.0 F8:50 NXB GRT I:10.4 24980 MOV 2498.0 F8:50 BND EOR
%   I:10.4  TT_7044  "TT-7044 ANALOG IN" %
%   F8:50  TT_7044_SCI  "TT-7044 SCALED INPUT" %
% Rung: 53 %
SOR BST SCP I:10.5 -4540.0 24980.0 -454.0 2498.0 F8:51 NXB LES I:10.5 -4540 MOV -454.0 F8:51 NXB GRT I:10.5 24980 MOV 2498.0 F8:51 BND EOR
%   I:10.5  TT_7045  "TT-7045 ANALOG IN" %
%   F8:51  TT_7045_SCI  "TT-7045 SCALED INPUT" %

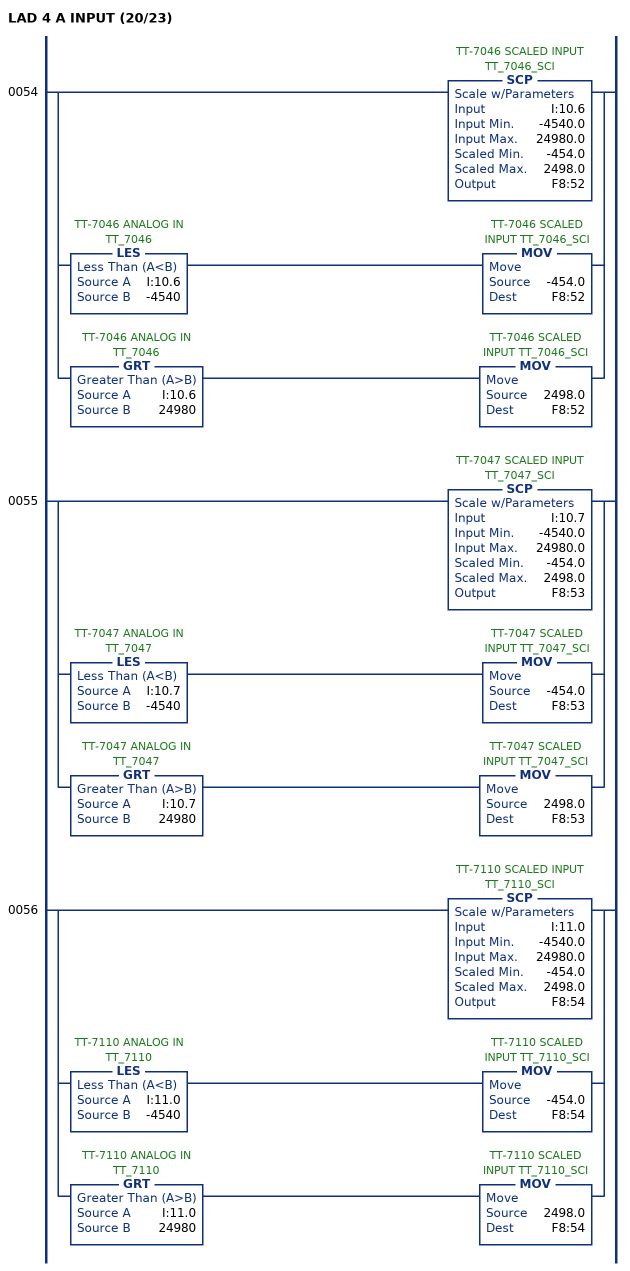
% Rung: 54 %
SOR BST SCP I:10.6 -4540.0 24980.0 -454.0 2498.0 F8:52 NXB LES I:10.6 -4540 MOV -454.0 F8:52 NXB GRT I:10.6 24980 MOV 2498.0 F8:52 BND EOR
%   I:10.6  TT_7046  "TT-7046 ANALOG IN" %
%   F8:52  TT_7046_SCI  "TT-7046 SCALED INPUT" %
% Rung: 55 %
SOR BST SCP I:10.7 -4540.0 24980.0 -454.0 2498.0 F8:53 NXB LES I:10.7 -4540 MOV -454.0 F8:53 NXB GRT I:10.7 24980 MOV 2498.0 F8:53 BND EOR
%   I:10.7  TT_7047  "TT-7047 ANALOG IN" %
%   F8:53  TT_7047_SCI  "TT-7047 SCALED INPUT" %
% Rung: 56 %
SOR BST SCP I:11.0 -4540.0 24980.0 -454.0 2498.0 F8:54 NXB LES I:11.0 -4540 MOV -454.0 F8:54 NXB GRT I:11.0 24980 MOV 2498.0 F8:54 BND EOR
%   I:11.0  TT_7110  "TT-7110 ANALOG IN" %
%   F8:54  TT_7110_SCI  "TT-7110 SCALED INPUT" %

